// LS Electric XG5000 project: 7_모타수증가
// PLC NewPLC
// module base 0 slot 0: 입출력 모듈:XBC-DR20S (DC 24V 입력 12점, 릴레이 출력 8점)

PROGRAM NewProgram (task: 스캔 프로그램)

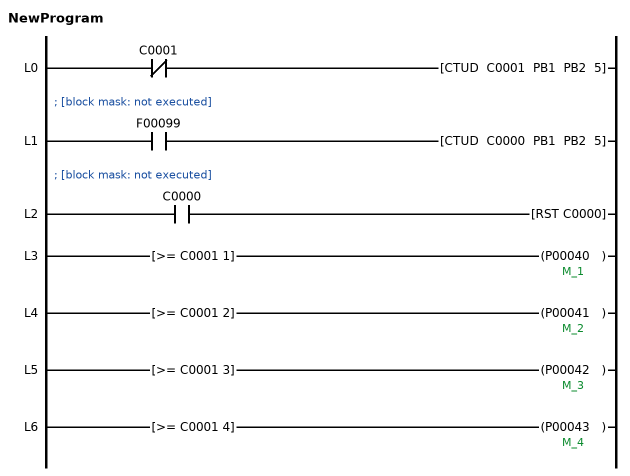
; L0
LOAD NOT  C0001
CTUD      C0001 PB1 PB2 5
; L1 (block mask: not executed)
LOAD      F00099
CTUD      C0000 PB1 PB2 5
; L2 (block mask: not executed)
LOAD      C0000
RST       C0000
; L3
LOAD>=    C0001 1
OUT       P00040	// M_1
; L4
LOAD>=    C0001 2
OUT       P00041	// M_2
; L5
LOAD>=    C0001 3
OUT       P00042	// M_3
; L6
LOAD>=    C0001 4
OUT       P00043	// M_4

VARIABLES AND COMMENTS (devices not used above)
P00000	BIT	PB1
P00001	BIT	PB2